(* Logix 5000 project; controller CLX_PCON Emulate 5570 rev 20.12; software revision 20.01 *)

TASK T01_Scan_10ms (periodic, rate 10 ms, priority 3, watchdog 500 ms) : P00_SUPPORT_FUNCTIONS
TASK T10_Scan_100ms (periodic, rate 100 ms, priority 5, watchdog 500 ms) : FAN_SIMULATOR

MODULES
   Local : Emulate 5570 (ICP 3, rev 20.12)
END_MODULES

TYPE PLC_DATIME :   // PLC Date and Time Basic Structure
STRUCT
   YEAR : DINT;
   MONTH : DINT;
   DAY : DINT;
   HOUR : DINT;
   MINUTE : DINT;
   SECOUND : DINT;
   uSECOND : DINT;
END_STRUCT
END_TYPE

TYPE STRG_DATIME :   // Date and Time String Format Basic Structure
STRUCT
   YEAR : STRING;
   MONTH : STRING;
   DAY : STRING;
   HOUR : STRING;
   MINUTE : STRING;
   SECOND : STRING;
   FDATE : STRING;   // FORMATTED DATE [YYYY/MM/DD]
   FTIME : STRING;   // FORMATTED TIME [HH:MM:SS]
END_STRUCT
END_TYPE

TYPE SUPPORT :   // Support Functions [Global Application]
STRUCT
   Log1 : BOOL;   // Logical 1: Always True
   Log0 : BOOL;   // Logical 0: Always False
   Ini : BOOL;   // Initialization Bit Pulse First Scan
   _2xHz : BOOL;   // Flash Bit 2 Hz Cycle 0.5 Sec Cycle
   _1xHz : BOOL;   // Flash Bit 1 Hz Cycle 1 Sec Cycle
   _05Hz : BOOL;   // Flash Bit 1/2 Hz Cycle 2 Sec Cycle
   Step_1x30 : INT;   // Base Counter 1 = [30ms/Count]
   Step_1x50 : INT;   // Base Counter 1 = [50ms/Count]
   Step_1x100 : INT;   // Base Counter 1 = [100ms/Count]
   Step_1x200 : INT;   // Base Counter 1 = [200ms/Count]
   Step_1x500 : INT;   // Base Counter 1 = [500ms/Count]
   Step_1x1000 : INT;   // Base Counter 1 = [1sec/Count]
   Beacon : SINT;   // Beacon Time Pulse
   Watchdog : INT;   // Communication Watchdog
   CSSG : DINT[5];   // Application Commissioning Flags [Miscellaneous]
END_STRUCT
END_TYPE

ADD_ON_INSTRUCTION RAMP   (* revision 1.0, vendor PTUS *)
// SPEED REFERENCE
VAR_INPUT
   X : REAL; {required}   // INPUT SPEED VALUE
   ACCELERATION : REAL; {visible}   // ACCELERATION RATE
   DECELERATION : REAL; {visible}   // DECELERATION RATE
   JERK : REAL; {visible}   // JERK RATE
END_VAR
VAR_OUTPUT
   Q : REAL; {access Read Only, required}   // OUTPUT SPEED REFERENCE [RAMPED]
END_VAR
VAR_INPUT
   RESET : BOOL; {required}   // RESET OUTPUT INITIALIZE TO ZERO
END_VAR
VAR
   SRAMP : S_CURVE := (RTSTime := 1); {access None}
END_VAR

ROUTINE Logic   (* structured text *)
// SPEED REFERENCE
   /////////////////////////////////////////////////////////////////////////////////////////////////////////////////////////
   // VERSION: 1.0 	DEVELOPER: ALEJANDRO CADENA			FUNCTION: SPEED CONTROL (RAMP) 			RELEASE: 10.27.2020	   //
   /////////////////////////////////////////////////////////////////////////////////////////////////////////////////////////
   // DESCRIPTION:	 																									   //
   //	THE FUNCTION PROVIDES A SMOOTH SPEED REFERENCE TO CONTROL A MOTION BY THE USE OF  A S-CURVE RAMP.				   //
   // 																													   //
   /////////////////////////////////////////////////////////////////////////////////////////////////////////////////////////
   
   //***********************************************************************************************************************
   // RAMP FUNCTION SETTINGS
   //***********************************************************************************************************************
   	SRAMP.In:= X;
   	SRAMP.AccelRate:= ACCELERATION;
   	SRAMP.DecelRate:= DECELERATION;
   	SRAMP.JerkRate:= JERK;
   	SRAMP.Initialize:= RESET;
   	SRAMP.InitialValue:= 0.0;
   
   //***********************************************************************************************************************
   // RAMP INTERNAL FUNCTION
   //***********************************************************************************************************************
   	SCRV(SRAMP);
   
   //***********************************************************************************************************************
   // FUNCTION OUTPUT
   //***********************************************************************************************************************
   	Q:= SRAMP.Out;
   
   //***********************************************************************************************************************
   // END OF SUBROUTINE
   //***********************************************************************************************************************
END_ROUTINE
END_ADD_ON_INSTRUCTION

ADD_ON_INSTRUCTION SPL_FAN   (* revision 1.0, vendor ODAN *)
VAR_INPUT
   SPEED : REAL; {required}   // ACTUAL FAN SPEED [RPM]
   NOM_PRESS : REAL; {required}   // PRESSURE AT NOMINAL POINT [EU]
   NOM_FLOW : REAL; {required}   // AIR FLOW AT NOMINAL POINT [EU]
   NOM_MOTOR : REAL; {required}   // MOTOR SPEED AT NOMINAL POINT [RPM]
   P_RATIO : REAL := 1.37;   // PRESSURE RATIO P0/P-NOM
   P_UL : REAL := 1000.0;   // PRESSURE UPPER LIMIT [OUTPUT]
   P_LL : REAL;   // PRESSURE LOWER LIMIT [OUTPUT]
   SCAN : INT := 10;   // SCAN [ms]
   TAU : INT := 50;   // TIME CONSTANT FILTER
END_VAR
VAR_OUTPUT
   PRSS : REAL; {access Read Only}   // PRESSURE [SIMULATED VALUE]
END_VAR
VAR
   Yn : REAL; {access None}   // PREVIOUS OUTPUT
   Y : REAL; {access None}   // FILTER OUTPUT
   X : REAL; {access None}   // FILTER INPUT
   TAUX : REAL; {access None}   // TIME CONSTANT AUX
   T_RATIO : REAL; {access None}   // TIME RATIO SCAN/TAU
   CF : REAL; {access None}   // FAN CURVE C-CONSTANT
   AF : REAL; {access None}   // FAN CURVE A-CONSTANT
   S_RATIO : REAL; {access None}   // SPEED RATIO
   AX : REAL; {access None}   // ADJUSTED CURVE A-CONSTANT
END_VAR

ROUTINE Logic   (* structured text *)
   ///////////////////////////////////////////////////////////////////////////////
   //SIMULATION PROCESS LIBRARY: FAN                     			VERSION: 1.0
   ///////////////////////////////////////////////////////////////////////////////
   //DEVELOPER: ALEJANDRO CADENA                     			RELEASE: 05.22.2021
   //
   //DESCRIPTION: THE FUNCTION SIMULATES THE STATIC PRESSURE CREATED BY A FAN
   //THE PRESSURE IS CALCULATED USING THE AFFINITY LAW (H1/H2) = (N1/N2)^2
   ///////////////////////////////////////////////////////////////////////////////
   
   //****************************************************************************
   // FAN CURVE CONSTANTS CALCULATION
   //****************************************************************************
    AF:= P_RATIO * NOM_PRESS;
   
    IF NOM_FLOW = 0.0 THEN
   
   	NOM_FLOW:= 1000;
   
    END_IF;		//END NOMINAL FLOW VALIDATION
   
    CF:= (AF - NOM_PRESS)/(NOM_FLOW * NOM_FLOW);
   
   //****************************************************************************
   // ADJUSTED CURVE CONSTANT CALCULATION
   //****************************************************************************
   	S_RATIO:= SPEED/NOM_MOTOR;
   
   	AX:= AF * (S_RATIO * S_RATIO);
   
   //****************************************************************************
   // INSTANTANEOUS STATIC PRESSURE CALCULATION
   //****************************************************************************
   	X:= AX - (CF * (NOM_FLOW * NOM_FLOW));
   
   //****************************************************************************
   // FIRST-ORDER-FILTER TIME CONSTANT VALIDATION
   //****************************************************************************
    IF TAU > SCAN THEN
   
    	TAUX:= TAU;
   
    ELSE
   
    	TAUX:= SCAN;
   
    END_IF;	//END TIME CONSTANT VALIDATION
   
   //****************************************************************************
   // FIRST-ORDER-FILTER PRESSURE ESTIMATION
   //****************************************************************************
    T_RATIO:= SCAN/TAUX;
   
    Y:= Yn + T_RATIO * (X - Yn);
   
   //****************************************************************************
   // STATIC PRESSURE OUTPUT VALUE
   //****************************************************************************
    IF Y > P_UL THEN
   
    	PRSS:= P_UL;
   
    ELSIF Y < P_LL THEN
   
    	PRSS:= P_LL;
   
    ELSE
   
   	PRSS:= Y;
   
    END_IF;	//END SET PRESSURE CALCULATION & VALIDATION
   
   //****************************************************************************
   // STATIC PRESSURE VALUE MEMORIZED
   //****************************************************************************
    Yn:= Y;
   
   //****************************************************************************
   // END OF SUBROUTINE
   //****************************************************************************
END_ROUTINE
END_ADD_ON_INSTRUCTION

VAR_GLOBAL   (* controller tags *)
   APP : SUPPORT := (Log1 := 1, _2xHz := 1, Step_1x30 := 12013, Step_1x50 := 654, Step_1x100 := 327, Step_1x200 := 16547, Step_1x500 := 6618, Step_1x1000 := 3309, Beacon := 1, Watchdog := 19808, CSSG[0] := -2147483648);
        .BEACON.0   // Support Functions [Global Application] Beacon Time Pulse 1 Second
        .BEACON.1   // Support Functions [Global Application] Beacon Time Pulse 1 Minute
        .BEACON.2   // Support Functions [Global Application] Beacon Time Pulse 1 Hour
        .CSSG[0].30   // PIC01 STEP TEST TUNING PROCEDURE [START COMMAND]
        .CSSG[0].11   // PIC01 MANUAL SELECTION [MANUAL COMMAND]
        .CSSG[0].10   // PIC01 AUTOMATIC SELECTION [MANUAL COMMAND]
        .CSSG[0].31   // PIC01 SETPOINT TEST TUNING PROCEDURE [START COMMAND]
   DUCT_PRESSURE : REAL := 800.00073;   // DUCT STATIC PRESSURE MEASUREMENT [mm H2O]
   N_REF : REAL := 1563.3318;   // FAN SPEED REFERENCE [RPM]
   PLC_CLK : PLC_DATIME := (YEAR := 2021, MONTH := 5, DAY := 25, HOUR := 14, MINUTE := 53, SECOUND := 11, uSECOND := 338360);   // EAF PLC ACTUAL CLOCK DATE AND TIME
   PLC_DTM : STRG_DATIME := (YEAR := '2021', MONTH := '05', DAY := '25', HOUR := '14', MINUTE := '53', SECOND := '10', FDATE := '2021/05/25', FTIME := '14:53:10');   // EAF PLC ACTUAL CLOCK DATE AND TIME [STRING FORMAT]
   VFD_SPEED : REAL := 1563.3318;   // VFD SPEED REFERENCE [RPM]
END_VAR

PROGRAM FAN_SIMULATOR   (* main routine A00_COMMON *)
VAR
   FAN : SPL_FAN := (SPEED := 1563.3318, NOM_PRESS := 1224.0, NOM_FLOW := 9400.0, NOM_MOTOR := 1800.0, P_RATIO := 1.41, P_UL := 1500.0, SCAN := 100, TAU := 400, PRSS := 800.00073);   // FAN [SIMULATOR]
END_VAR

ROUTINE A00_COMMON   (* ladder *)
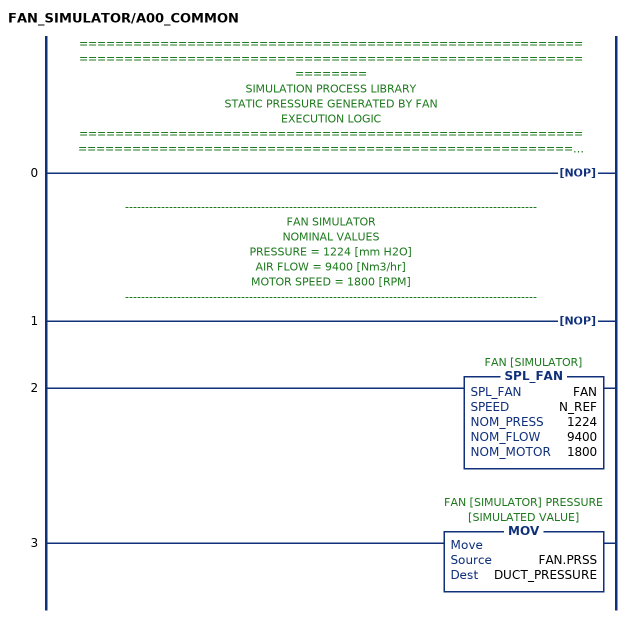
   // ========================================================================================================================
   // SIMULATION PROCESS LIBRARY
   // STATIC PRESSURE GENERATED BY FAN
   // EXECUTION LOGIC
   // ========================================================================================================================
   0: NOP();
   // -------------------------------------------------------------------------------------------------------
   // FAN SIMULATOR
   // NOMINAL VALUES
   // PRESSURE = 1224 [mm H2O]
   // AIR FLOW = 9400 [Nm3/hr]
   // MOTOR SPEED = 1800 [RPM]
   // -------------------------------------------------------------------------------------------------------
   1: NOP();
   2: SPL_FAN(FAN,N_REF,1224,9400,1800);
   3: MOV(FAN.PRSS,DUCT_PRESSURE);
END_ROUTINE
END_PROGRAM

PROGRAM P00_SUPPORT_FUNCTIONS   (* main routine A00_COMMON *)
VAR
   APP_CNT : DINT[20] := ([0] := 32, [1] := 16275, [2] := 1, [3] := 56, [4] := 3, [5] := 3, [6] := 3, [8] := 43, [10] := 43, [11] := 23, [12] := 48);
        [2]   // Auxiliary Counter Rate: 10ms/Per Count [30 ms]
        [11]   // Auxiliary Counter Acc: 1Sec/Per Count
        [12]   // Auxiliary Counter Acc: 1Min/Per Count
        [0]   // Auxiliary Counter Rate: 10ms/Per Count [10 ms]
        [1]   // Auxiliary Counter Rate: 10ms/Per Count [20 ms]
        [3]   // Auxiliary Counter Rate: 10ms/Per Count [40 ms]
        [4]   // Auxiliary Counter Rate: 10ms/Per Count [50 ms]
        [5]   // Auxiliary Counter Rate: 10ms/Per Count [100 ms]
        [6]   // Auxiliary Counter Rate: 10ms/Per Count [200 ms]
        [7]   // Auxiliary Counter Rate: 10ms/Per Count [300 ms]
        [8]   // Auxiliary Counter Rate: 10ms/Per Count [500 ms]
        [10]   // Auxiliary Counter Rate: 10ms/Per Count [1000 ms]
   APP_FLG : DINT := -2147483648;
        .10   // TICK PULSE [1 SEC]
        .0   // TICK PULSE [10 MSEC]
        .1   // TICK PULSE [20 MSEC]
        .2   // TICK PULSE [30 MSEC]
        .5   // TICK PULSE [100 MSEC]
        .3   // TICK PULSE [40 MSEC]
        .4   // TICK PULSE [50 MSEC]
        .7   // TICK PULSE [300 MSEC]
        .6   // TICK PULSE [200 MSEC]
        .11   // TICK PULSE [1 MIN]
        .12   // TICK PULSE [1 HR]
        .30   // CLOCK READ ASSIGN FORMAT TO DATE AND TIME [PULSE]
        .8   // TICK PULSE [500 MSEC]
   APP_ONS : DINT := 1073741832;
   APP_TMR : TIMER[30] := ([0].PRE := 1000, [0].ACC := 1000, [1].PRE := 999, [1].ACC := 141, [1].EN := 1, [1].TT := 1, [2].PRE := 999, [3].PRE := 1999, [3].ACC := 1181, [3].EN := 1, [3].TT := 1, [4].PRE := 1999, [5].PRE := 600, [5].ACC := 420, [5].TT := 1, [5].DN := 1, [6].PRE := 600, [6].ACC := 611, [7].PRE := 600, [7].ACC := 600, [10].PRE := 500, [10].ACC := 500, [10].EN := 1, [10].DN := 1, [11].PRE := 500, [11].ACC := 490, [11].EN := 1, [11].TT := 1);
        [0]   // Initialization Bit First Scan Pulse - Time Control [Delay]
        [10]   // Flash Timer Duty Cycle On [0.5 Sec]
        [11]   // Flash Timer Duty Cycle Off [0.5 Sec]
        [1]   // Flash Timer Duty Cycle On [1 Sec]
        [2]   // Flash Timer Duty Cycle Off [1 Sec]
        [3]   // Flash Timer Duty Cycle On [2 Sec]
        [4]   // Flash Timer Duty Cycle Off [2 Sec]
        [5]   // Beacon Time Pulse 1 Second [TIMER]
        [6]   // Beacon Time Pulse 1 Minute [TIMER]
        [7]   // Beacon Time Pulse 1 Hour [TIMER]
   DT_COLON : STRING := ':';
   DT_SLASH : STRING := '/';
   DT_ZERO : STRING := '0';
   SIMULATION_ON : BOOL;   // APPLICATION BASIC SIMULATION ENABLE MANUAL COMMAND
END_VAR

ROUTINE A00_COMMON   (* ladder *)
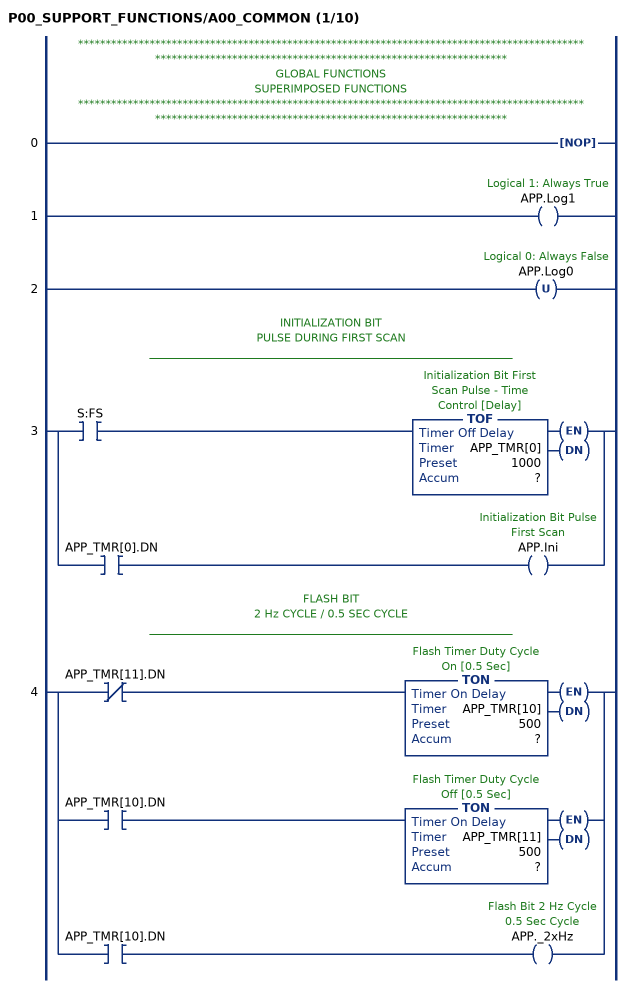
   // ************************************************************************************************************************************************************
   // GLOBAL FUNCTIONS
   // SUPERIMPOSED FUNCTIONS
   // ************************************************************************************************************************************************************
   0: NOP();
   1: OTE(APP.Log1);
   2: OTU(APP.Log0);
   // INITIALIZATION BIT
   // PULSE DURING FIRST SCAN
   // __________________________________________________________________
   3: [XIC(S:FS) TOF(APP_TMR[0],?,?) ,XIC(APP_TMR[0].DN) OTE(APP.Ini) ];
   // FLASH BIT
   // 2 Hz CYCLE / 0.5 SEC CYCLE
   // __________________________________________________________________
   4: [XIO(APP_TMR[11].DN) TON(APP_TMR[10],?,?) ,XIC(APP_TMR[10].DN) TON(APP_TMR[11],?,?) ,XIC(APP_TMR[10].DN) OTE(APP._2xHz) ];
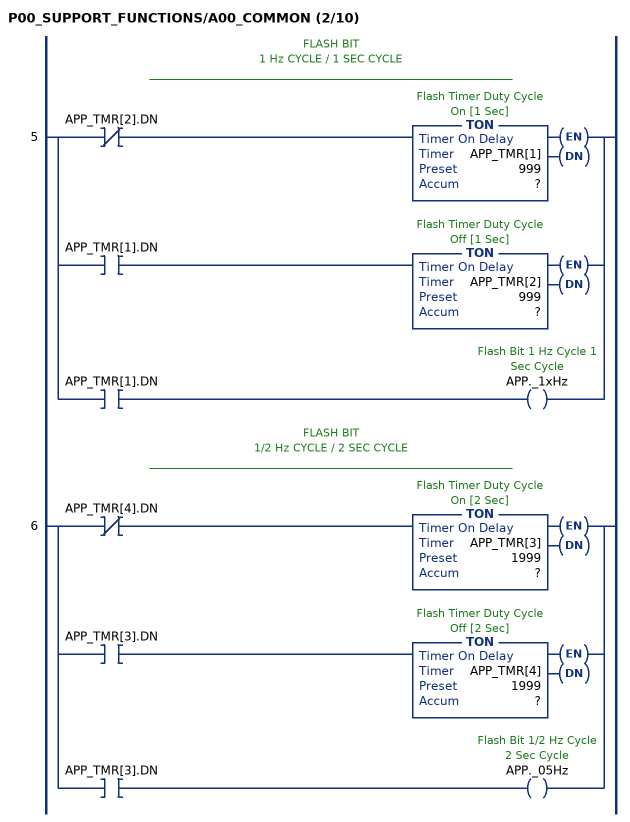
   // FLASH BIT
   // 1 Hz CYCLE / 1 SEC CYCLE
   // __________________________________________________________________
   5: [XIO(APP_TMR[2].DN) TON(APP_TMR[1],?,?) ,XIC(APP_TMR[1].DN) TON(APP_TMR[2],?,?) ,XIC(APP_TMR[1].DN) OTE(APP._1xHz) ];
   // FLASH BIT
   // 1/2 Hz CYCLE / 2 SEC CYCLE
   // __________________________________________________________________
   6: [XIO(APP_TMR[4].DN) TON(APP_TMR[3],?,?) ,XIC(APP_TMR[3].DN) TON(APP_TMR[4],?,?) ,XIC(APP_TMR[3].DN) OTE(APP._05Hz) ];
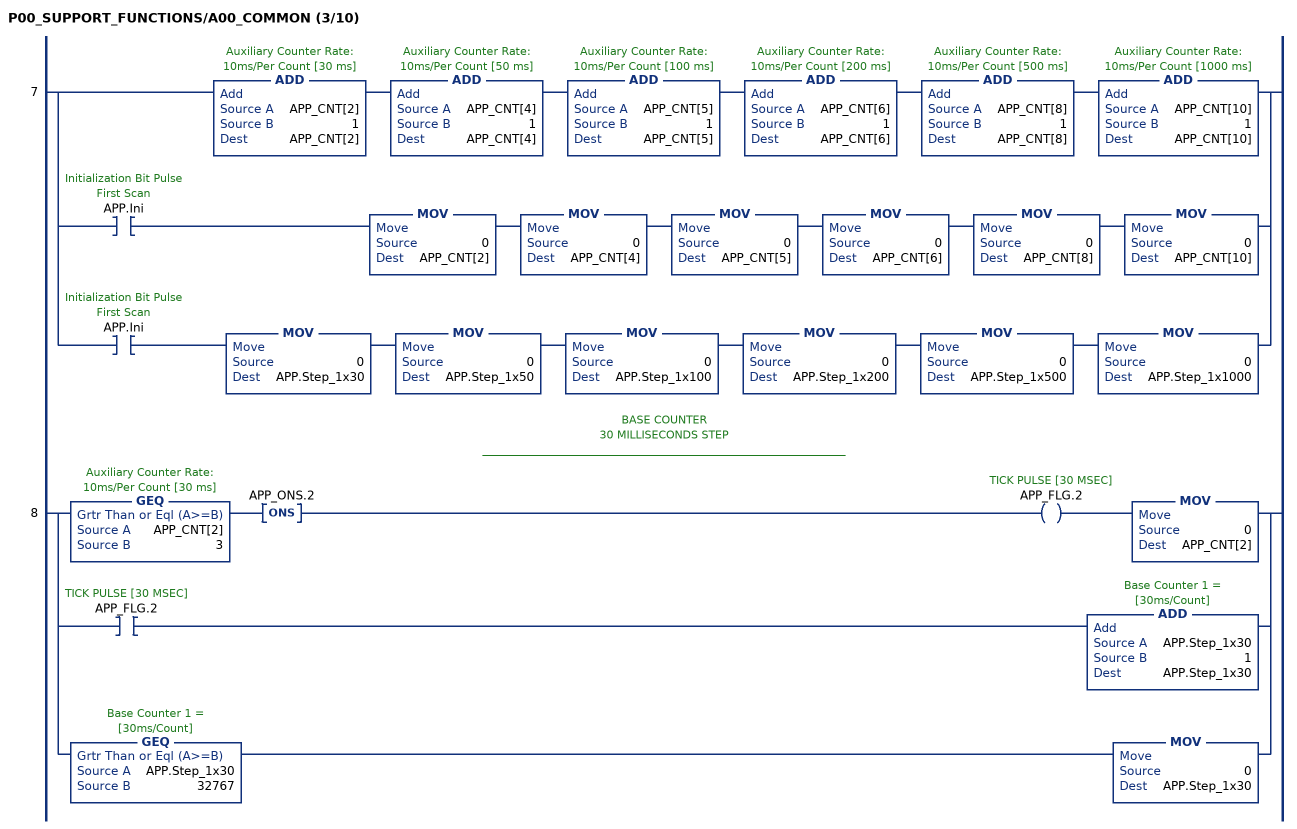
   7: [ADD(APP_CNT[2],1,APP_CNT[2]) ADD(APP_CNT[4],1,APP_CNT[4]) ADD(APP_CNT[5],1,APP_CNT[5]) ADD(APP_CNT[6],1,APP_CNT[6]) ADD(APP_CNT[8],1,APP_CNT[8]) ADD(APP_CNT[10],1,APP_CNT[10]) ,XIC(APP.Ini) MOV(0,APP_CNT[2]) MOV(0,APP_CNT[4]) MOV(0,APP_CNT[5]) MOV(0,APP_CNT[6]) MOV(0,APP_CNT[8]) MOV(0,APP_CNT[10]) ,XIC(APP.Ini) MOV(0,APP.Step_1x30) MOV(0,APP.Step_1x50) MOV(0,APP.Step_1x100) MOV(0,APP.Step_1x200) MOV(0,APP.Step_1x500) MOV(0,APP.Step_1x1000) ];
   // BASE COUNTER
   // 30 MILLISECONDS STEP
   // __________________________________________________________________
   8: [GEQ(APP_CNT[2],3) ONS(APP_ONS.2) OTE(APP_FLG.2) MOV(0,APP_CNT[2]) ,XIC(APP_FLG.2) ADD(APP.Step_1x30,1,APP.Step_1x30) ,GEQ(APP.Step_1x30,32767) MOV(0,APP.Step_1x30) ];
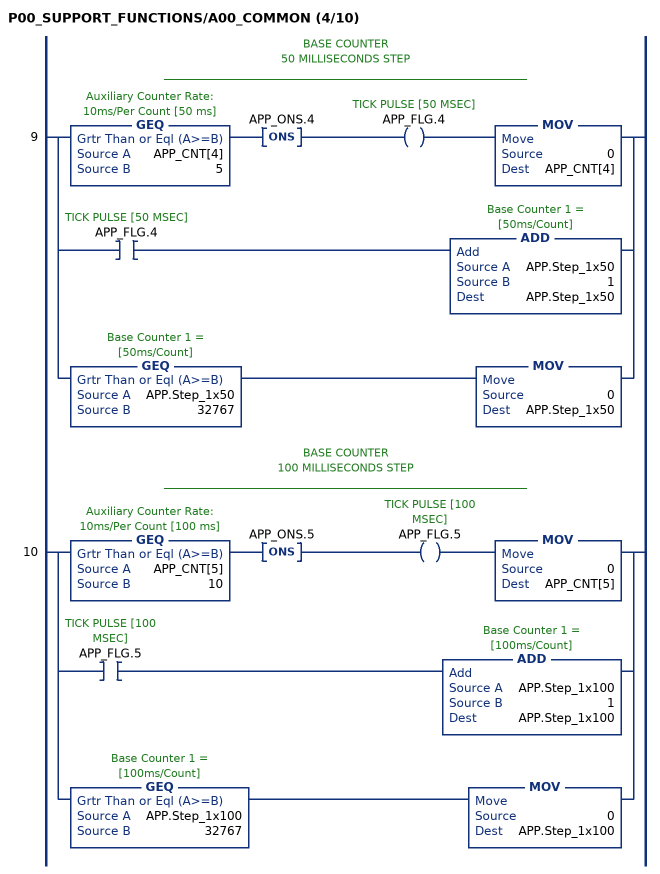
   // BASE COUNTER
   // 50 MILLISECONDS STEP
   // __________________________________________________________________
   9: [GEQ(APP_CNT[4],5) ONS(APP_ONS.4) OTE(APP_FLG.4) MOV(0,APP_CNT[4]) ,XIC(APP_FLG.4) ADD(APP.Step_1x50,1,APP.Step_1x50) ,GEQ(APP.Step_1x50,32767) MOV(0,APP.Step_1x50) ];
   // BASE COUNTER
   // 100 MILLISECONDS STEP
   // __________________________________________________________________
   10: [GEQ(APP_CNT[5],10) ONS(APP_ONS.5) OTE(APP_FLG.5) MOV(0,APP_CNT[5]) ,XIC(APP_FLG.5) ADD(APP.Step_1x100,1,APP.Step_1x100) ,GEQ(APP.Step_1x100,32767) MOV(0,APP.Step_1x100) ];
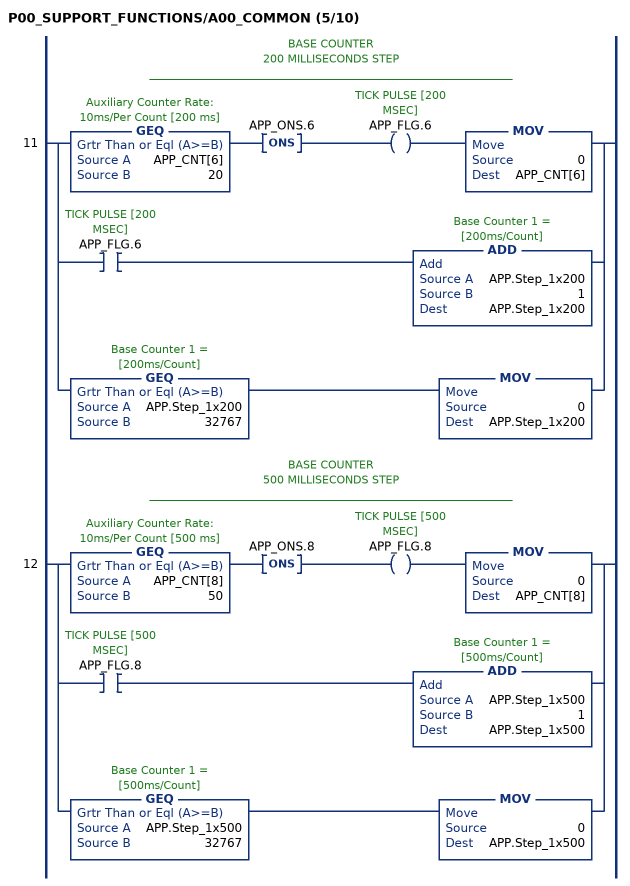
   // BASE COUNTER
   // 200 MILLISECONDS STEP
   // __________________________________________________________________
   11: [GEQ(APP_CNT[6],20) ONS(APP_ONS.6) OTE(APP_FLG.6) MOV(0,APP_CNT[6]) ,XIC(APP_FLG.6) ADD(APP.Step_1x200,1,APP.Step_1x200) ,GEQ(APP.Step_1x200,32767) MOV(0,APP.Step_1x200) ];
   // BASE COUNTER
   // 500 MILLISECONDS STEP
   // __________________________________________________________________
   12: [GEQ(APP_CNT[8],50) ONS(APP_ONS.8) OTE(APP_FLG.8) MOV(0,APP_CNT[8]) ,XIC(APP_FLG.8) ADD(APP.Step_1x500,1,APP.Step_1x500) ,GEQ(APP.Step_1x500,32767) MOV(0,APP.Step_1x500) ];
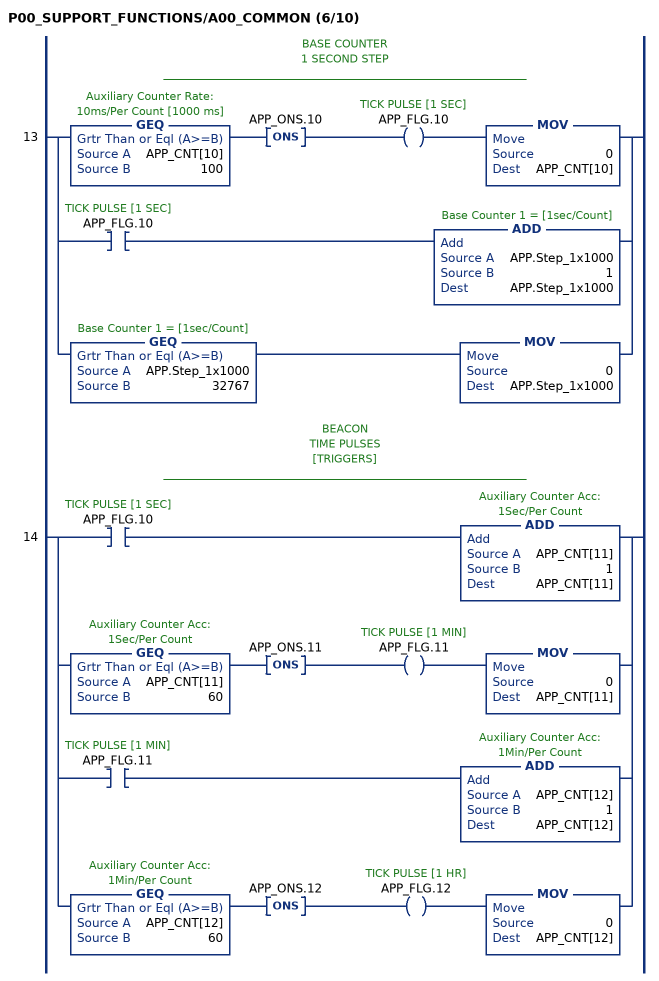
   // BASE COUNTER
   // 1 SECOND STEP
   // __________________________________________________________________
   13: [GEQ(APP_CNT[10],100) ONS(APP_ONS.10) OTE(APP_FLG.10) MOV(0,APP_CNT[10]) ,XIC(APP_FLG.10) ADD(APP.Step_1x1000,1,APP.Step_1x1000) ,GEQ(APP.Step_1x1000,32767) MOV(0,APP.Step_1x1000) ];
   // BEACON
   // TIME PULSES
   // [TRIGGERS]
   // __________________________________________________________________
   14: [XIC(APP_FLG.10) ADD(APP_CNT[11],1,APP_CNT[11]) ,GEQ(APP_CNT[11],60) ONS(APP_ONS.11) OTE(APP_FLG.11) MOV(0,APP_CNT[11]) ,XIC(APP_FLG.11) ADD(APP_CNT[12],1,APP_CNT[12]) ,GEQ(APP_CNT[12],60) ONS(APP_ONS.12) OTE(APP_FLG.12) MOV(0,APP_CNT[12]) ];
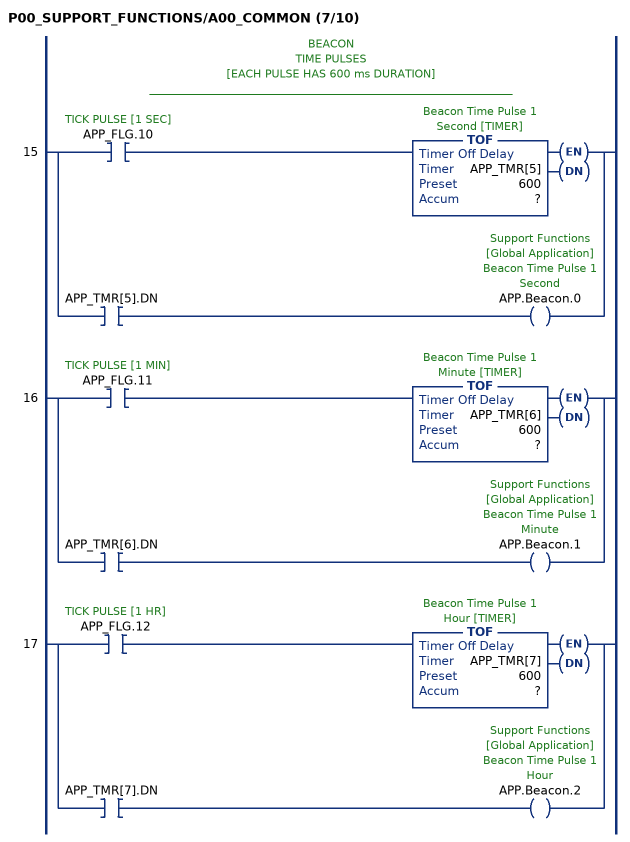
   // BEACON
   // TIME PULSES
   // [EACH PULSE HAS 600 ms DURATION]
   // __________________________________________________________________
   15: [XIC(APP_FLG.10) TOF(APP_TMR[5],?,?) ,XIC(APP_TMR[5].DN) OTE(APP.Beacon.0) ];
   16: [XIC(APP_FLG.11) TOF(APP_TMR[6],?,?) ,XIC(APP_TMR[6].DN) OTE(APP.Beacon.1) ];
   17: [XIC(APP_FLG.12) TOF(APP_TMR[7],?,?) ,XIC(APP_TMR[7].DN) OTE(APP.Beacon.2) ];
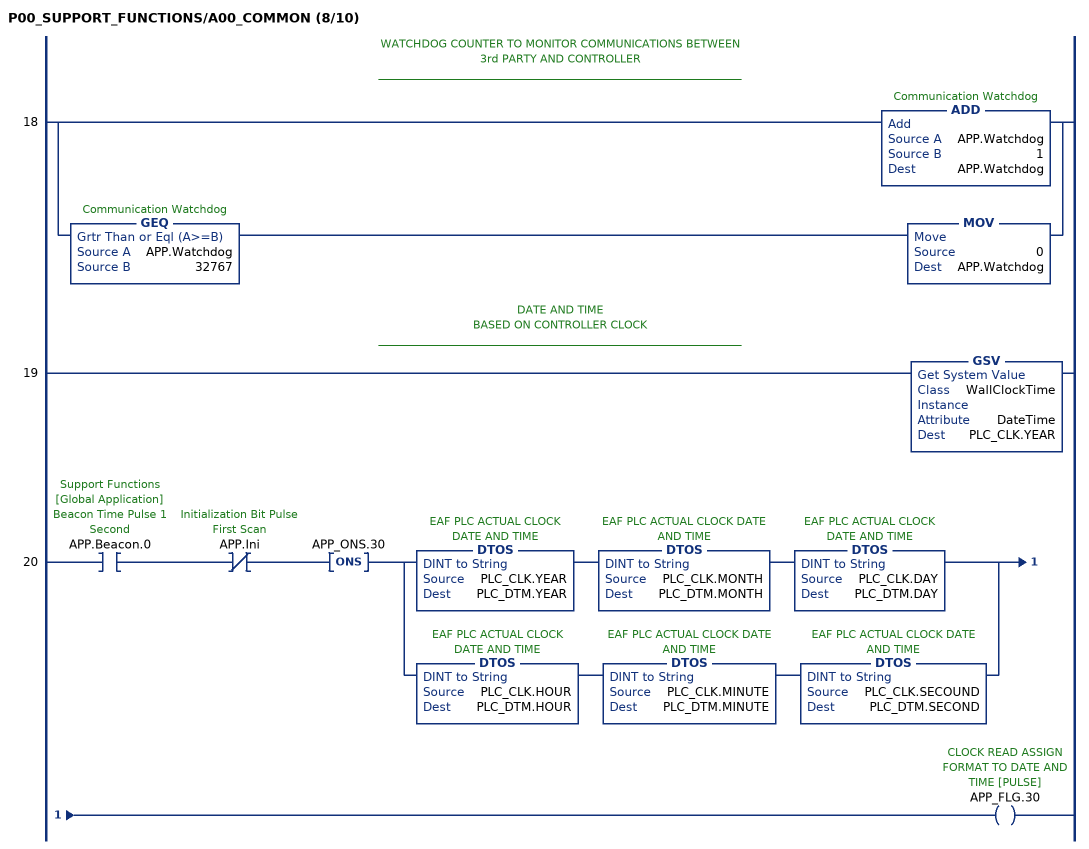
   // WATCHDOG COUNTER TO MONITOR COMMUNICATIONS BETWEEN
   // 3rd PARTY AND CONTROLLER
   // __________________________________________________________________
   18: [ADD(APP.Watchdog,1,APP.Watchdog) ,GEQ(APP.Watchdog,32767) MOV(0,APP.Watchdog) ];
   // DATE AND TIME
   // BASED ON CONTROLLER CLOCK
   // __________________________________________________________________
   19: GSV(WallClockTime,,DateTime,PLC_CLK.YEAR);
   20: XIC(APP.Beacon.0)XIO(APP.Ini)ONS(APP_ONS.30)[DTOS(PLC_CLK.YEAR,PLC_DTM.YEAR) DTOS(PLC_CLK.MONTH,PLC_DTM.MONTH) DTOS(PLC_CLK.DAY,PLC_DTM.DAY) ,DTOS(PLC_CLK.HOUR,PLC_DTM.HOUR) DTOS(PLC_CLK.MINUTE,PLC_DTM.MINUTE) DTOS(PLC_CLK.SECOUND,PLC_DTM.SECOND) ]OTE(APP_FLG.30);
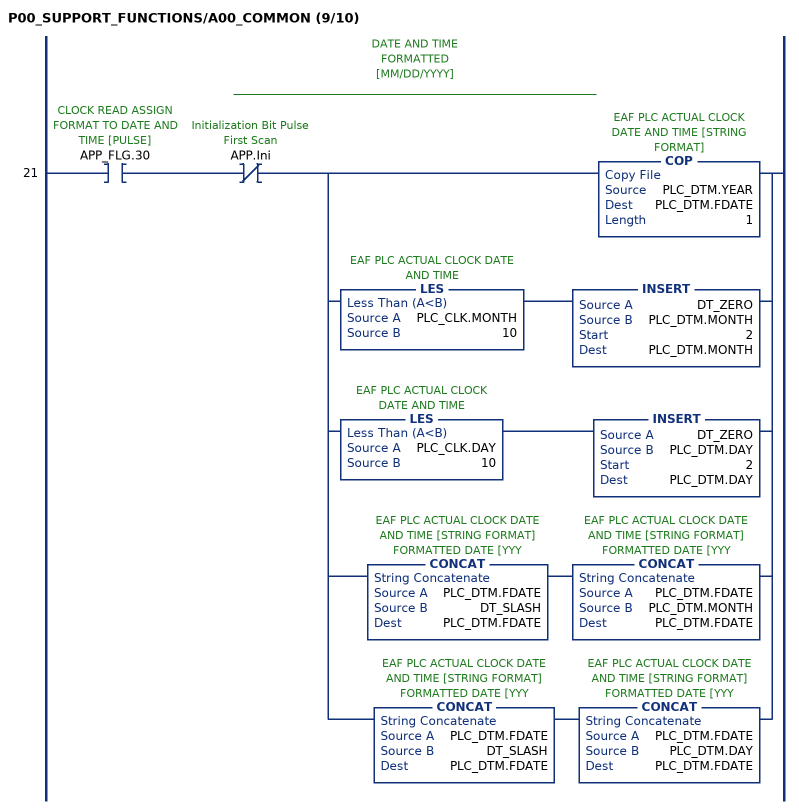
   // DATE AND TIME
   // FORMATTED
   // [MM/DD/YYYY]
   // __________________________________________________________________
   21: XIC(APP_FLG.30)XIO(APP.Ini)[COP(PLC_DTM.YEAR,PLC_DTM.FDATE,1) ,LES(PLC_CLK.MONTH,10) INSERT(DT_ZERO,PLC_DTM.MONTH,2,PLC_DTM.MONTH) ,LES(PLC_CLK.DAY,10) INSERT(DT_ZERO,PLC_DTM.DAY,2,PLC_DTM.DAY) ,CONCAT(PLC_DTM.FDATE,DT_SLASH,PLC_DTM.FDATE) CONCAT(PLC_DTM.FDATE,PLC_DTM.MONTH,PLC_DTM.FDATE) ,CONCAT(PLC_DTM.FDATE,DT_SLASH,PLC_DTM.FDATE) CONCAT(PLC_DTM.FDATE,PLC_DTM.DAY,PLC_DTM.FDATE) ];
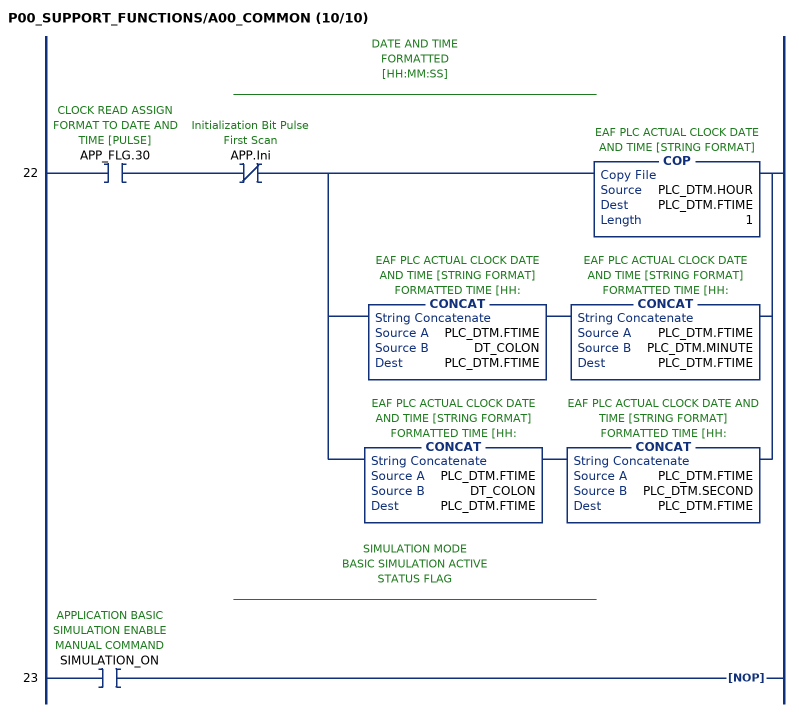
   // DATE AND TIME
   // FORMATTED
   // [HH:MM:SS]
   // __________________________________________________________________
   22: XIC(APP_FLG.30)XIO(APP.Ini)[COP(PLC_DTM.HOUR,PLC_DTM.FTIME,1) ,CONCAT(PLC_DTM.FTIME,DT_COLON,PLC_DTM.FTIME) CONCAT(PLC_DTM.FTIME,PLC_DTM.MINUTE,PLC_DTM.FTIME) ,CONCAT(PLC_DTM.FTIME,DT_COLON,PLC_DTM.FTIME) CONCAT(PLC_DTM.FTIME,PLC_DTM.SECOND,PLC_DTM.FTIME) ];
   // SIMULATION MODE
   // BASIC SIMULATION ACTIVE
   // STATUS FLAG
   // __________________________________________________________________
   23: XIC(SIMULATION_ON)NOP();
END_ROUTINE
END_PROGRAM

PROGRAM PRESSURE_CONTROL   (* main routine A00_COMMON *)
VAR
   FLAG : DINT[5];
        [0].30   // PIC01 STEP TEST TUNING PROCEDURE [START PULSE]
        [0].1   // PIC01 STEP TEST TUNING PROCEDURE [ACTIVE FLAG]
        [0].5   // PIC01 STEP TEST TUNING PROCEDURE [STEP APPLIED]
        [0].31   // PIC01 SETPOINT TEST TUNING PROCEDURE [START PULSE]
        [0].6   // PIC01 SETPONT TEST TUNING PROCEDURE [STEP APPLIED]
        [0].2   // PIC01 SETPOINT TEST TUNING PROCEDURE [ACTIVE FLAG]
   ONS : DINT[5] := ([0] := -2147483648);
   PIC01 : PID := (CTL := -2147449728, EN := 1, INI := 1, DVNA := 1, PVHA := 1, SP := 800.0, KP := 0.52, KI := 0.77, MAXS := 1800.0, SO := 86.85177, MAXO := 100.0, UPD := 0.1, PV := 800.00073, ERR := -0.0007324219, OUT := 86.85177, MAXI := 1800.0, MAXCV := 100.0, MAXTIE := 100.0, DATA[0] := 86.85179, DATA[1] := -711.11176, DATA[2] := 800.00073, DATA[3] := -0.0007324219, DATA[4] := 800.0, DATA[5] := 0.055555556, DATA[6] := 1.0, DATA[7] := 1.6, DATA[8] := 0.52, DATA[9] := 0.77, DATA[11] := 0.52, DATA[12] := 0.77, DATA[15] := 1.0, DATA[16] := 1.0);   // DUCT PRESSURE PIC01 CONTROLLER
   PIC01_MANUAL : REAL := 86.85177;
   PIC01_MODE : DINT := 1024;
        .1   // PIC01 PRESSURE CONTROL MANUAL MODE SELECTED [PULSE]
        .0   // PIC01 PRESSURE CONTROL AUTOMATIC MODE SELECTED [PULSE]
        .10   // PIC01 PRESSURE CONTROL AUTOMATIC MODE [ACTIVE]
        .11   // PIC01 PRESSURE CONTROL MANUAL MODE [ACTIVE]
   PIC01_REFERENCE : REAL := 86.85177;
   PIC01_SETPOINT : REAL := 800.0;
   TIMER : TIMER[10] := ([5].PRE := 40000, [6].PRE := 20000);
        [6]   // PIC01 SETPOINT TEST TUNING PROCEDURE STEP CHANGE [TIMER]
        [5]   // PIC01 STEP TEST TUNING PROCEDURE STEP CHANGE [TIMER]
   VFD_RAMP : RAMP := (X := 1563.3318, ACCELERATION := 300.0, DECELERATION := 300.0, JERK := 1000.0, Q := 1563.3318);   // VFD FAN RAMP SPEED TO DRIVE [RPM]
END_VAR

ROUTINE A00_COMMON   (* ladder *)
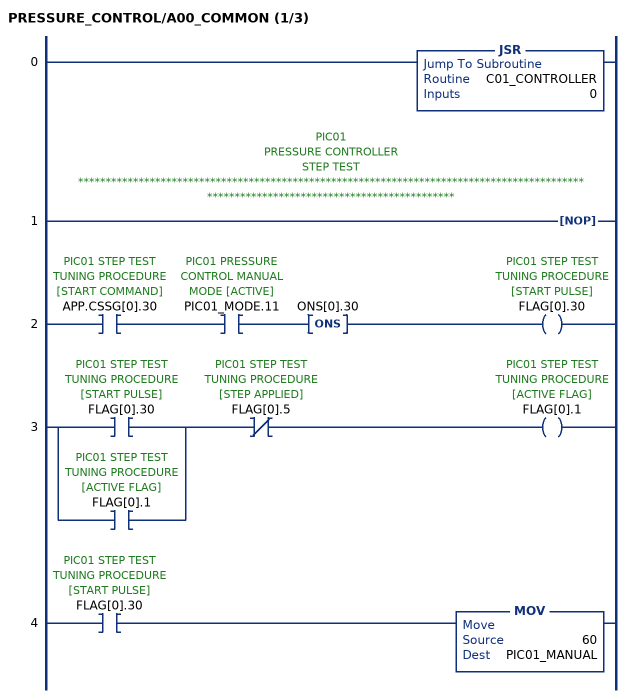
   0: JSR(C01_CONTROLLER,0);
   // PIC01
   // PRESSURE CONTROLLER
   // STEP TEST
   // *****************************************************************************************************************************************
   1: NOP();
   2: XIC(APP.CSSG[0].30)XIC(PIC01_MODE.11)ONS(ONS[0].30)OTE(FLAG[0].30);
   3: [XIC(FLAG[0].30) ,XIC(FLAG[0].1) ]XIO(FLAG[0].5)OTE(FLAG[0].1);
   4: XIC(FLAG[0].30)MOV(60,PIC01_MANUAL);
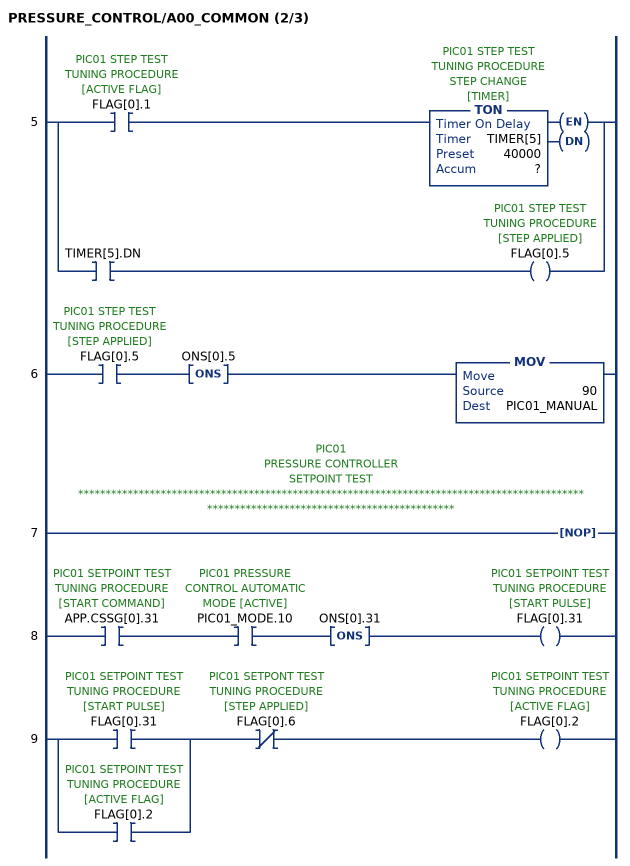
   5: [XIC(FLAG[0].1) TON(TIMER[5],?,?) ,XIC(TIMER[5].DN) OTE(FLAG[0].5) ];
   6: XIC(FLAG[0].5)ONS(ONS[0].5)MOV(90,PIC01_MANUAL);
   // PIC01
   // PRESSURE CONTROLLER
   // SETPOINT TEST
   // *****************************************************************************************************************************************
   7: NOP();
   8: XIC(APP.CSSG[0].31)XIC(PIC01_MODE.10)ONS(ONS[0].31)OTE(FLAG[0].31);
   9: [XIC(FLAG[0].31) ,XIC(FLAG[0].2) ]XIO(FLAG[0].6)OTE(FLAG[0].2);
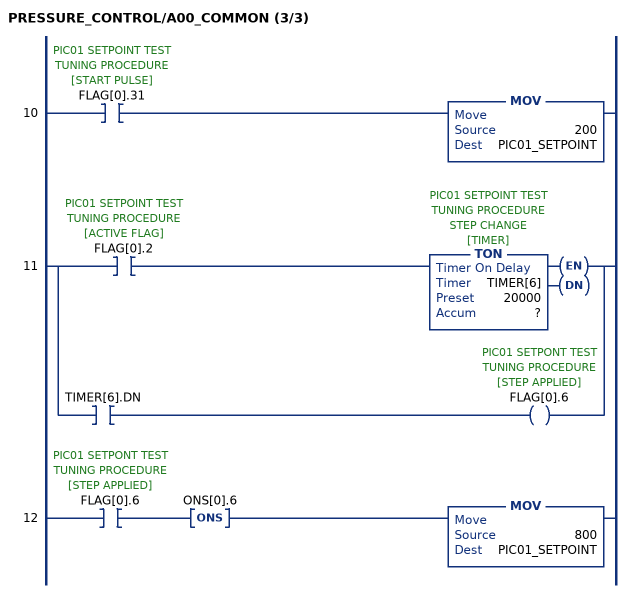
   10: XIC(FLAG[0].31)MOV(200,PIC01_SETPOINT);
   11: [XIC(FLAG[0].2) TON(TIMER[6],?,?) ,XIC(TIMER[6].DN) OTE(FLAG[0].6) ];
   12: XIC(FLAG[0].6)ONS(ONS[0].6)MOV(800,PIC01_SETPOINT);
END_ROUTINE

ROUTINE C01_CONTROLLER   (* ladder *)
// PRESSURE CONTROL
// PID CONTROLLER
// OPERATION AND CONTROL
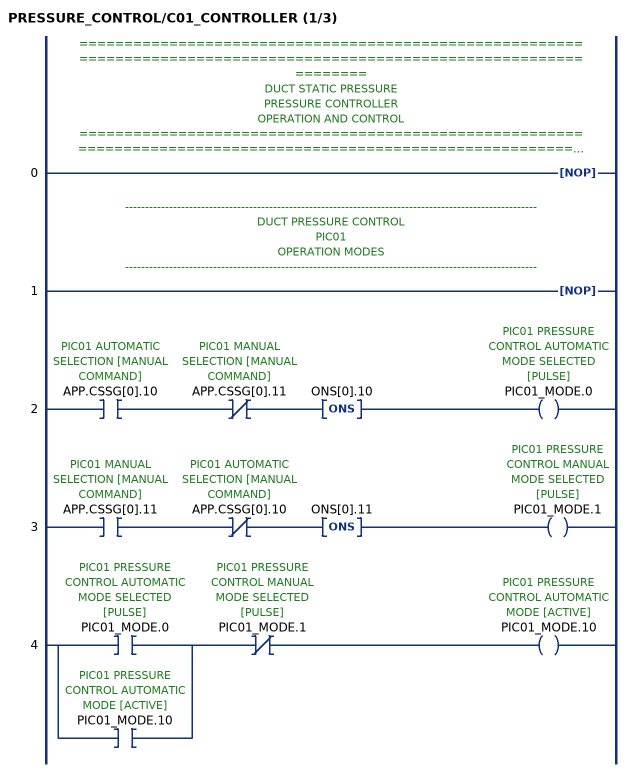
   // ========================================================================================================================
   // DUCT STATIC PRESSURE
   // PRESSURE CONTROLLER
   // OPERATION AND CONTROL
   // ========================================================================================================================
   0: NOP();
   // -------------------------------------------------------------------------------------------------------
   // DUCT PRESSURE CONTROL
   // PIC01
   // OPERATION MODES
   // -------------------------------------------------------------------------------------------------------
   1: NOP();
   2: XIC(APP.CSSG[0].10)XIO(APP.CSSG[0].11)ONS(ONS[0].10)OTE(PIC01_MODE.0);
   3: XIC(APP.CSSG[0].11)XIO(APP.CSSG[0].10)ONS(ONS[0].11)OTE(PIC01_MODE.1);
   4: [XIC(PIC01_MODE.0) ,XIC(PIC01_MODE.10) ]XIO(PIC01_MODE.1)OTE(PIC01_MODE.10);
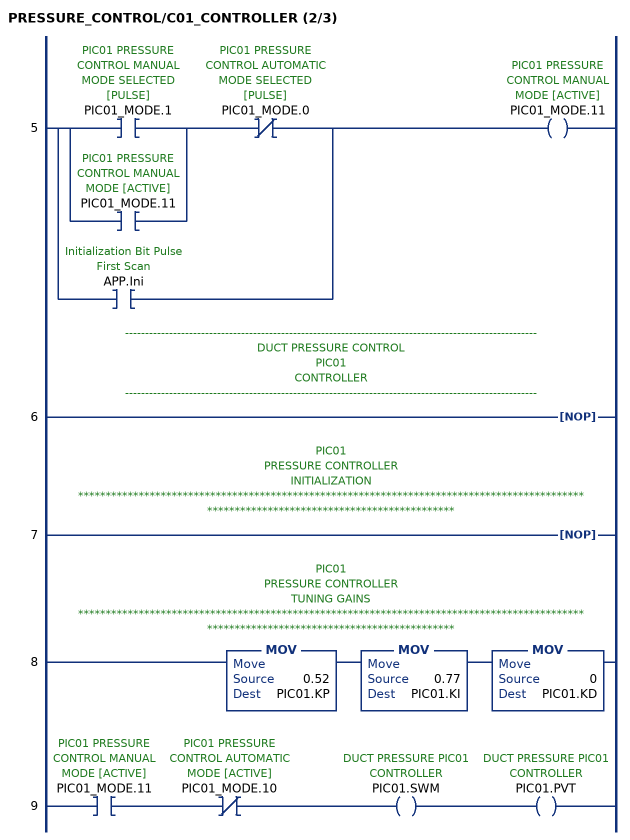
   5: [[XIC(PIC01_MODE.1) ,XIC(PIC01_MODE.11) ] XIO(PIC01_MODE.0) ,XIC(APP.Ini) ]OTE(PIC01_MODE.11);
   // -------------------------------------------------------------------------------------------------------
   // DUCT PRESSURE CONTROL
   // PIC01
   // CONTROLLER
   // -------------------------------------------------------------------------------------------------------
   6: NOP();
   // PIC01
   // PRESSURE CONTROLLER
   // INITIALIZATION
   // *****************************************************************************************************************************************
   7: NOP();
   // PIC01
   // PRESSURE CONTROLLER
   // TUNING GAINS
   // *****************************************************************************************************************************************
   8: MOV(0.52,PIC01.KP)MOV(0.77,PIC01.KI)MOV(0,PIC01.KD);
   9: XIC(PIC01_MODE.11)XIO(PIC01_MODE.10)OTE(PIC01.SWM)OTE(PIC01.PVT);
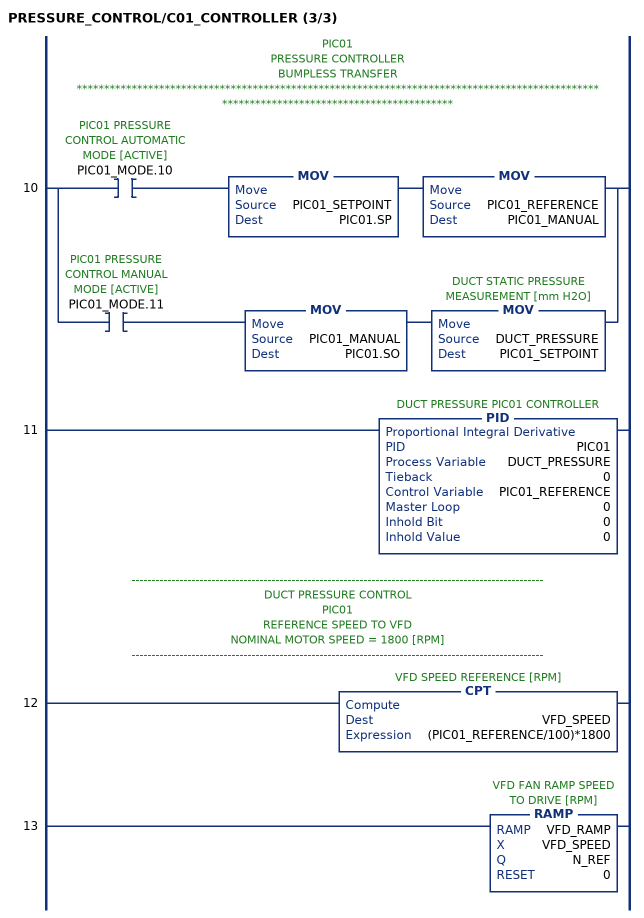
   // PIC01
   // PRESSURE CONTROLLER
   // BUMPLESS TRANSFER
   // *****************************************************************************************************************************************
   10: [XIC(PIC01_MODE.10) MOV(PIC01_SETPOINT,PIC01.SP) MOV(PIC01_REFERENCE,PIC01_MANUAL) ,XIC(PIC01_MODE.11) MOV(PIC01_MANUAL,PIC01.SO) MOV(DUCT_PRESSURE,PIC01_SETPOINT) ];
   11: PID(PIC01,DUCT_PRESSURE,0,PIC01_REFERENCE,0,0,0);
   // -------------------------------------------------------------------------------------------------------
   // DUCT PRESSURE CONTROL
   // PIC01
   // REFERENCE SPEED TO VFD
   // NOMINAL MOTOR SPEED = 1800 [RPM]
   // -------------------------------------------------------------------------------------------------------
   12: CPT(VFD_SPEED,(PIC01_REFERENCE/100)*1800);
   13: RAMP(VFD_RAMP,VFD_SPEED,N_REF,0);
END_ROUTINE
END_PROGRAM
